FUNCTION_BLOCK btb2
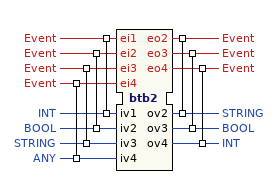
  EVENT_INPUT
    ei1 WITH iv1;
    ei2 WITH iv2;
    ei3 WITH iv3;
    ei4 WITH iv4;
  END_EVENT
  EVENT_OUTPUT
    eo2 WITH ov2;
    eo3 WITH ov3;
    eo4 WITH ov4;
  END_EVENT
  VAR_INPUT
    iv1 : INT;
    iv2 : BOOL;
    iv3 : STRING;
    iv4 : ANY;
  END_VAR
  VAR_OUTPUT
    ov2 : STRING;
    ov3 : BOOL;
    ov4 : INT;
  END_VAR
  EC_STATES
    START;
  END_STATES
END_FUNCTION_BLOCK
